TYPE typeMessage :
STRUCT
	//defines a list of messages to display for each type of message
	message: ARRAY [0..1000] OF BOOL;
	text:ARRAY[0..1000] of STRING(255);
END_STRUCT
END_TYPE

(* stored: Version 1.1.0.1, ProductVersion 3.1.4024.12
   DUT typeMessage: Id {221336c1-ab93-4c6c-ba86-6e53bedca566} *)
